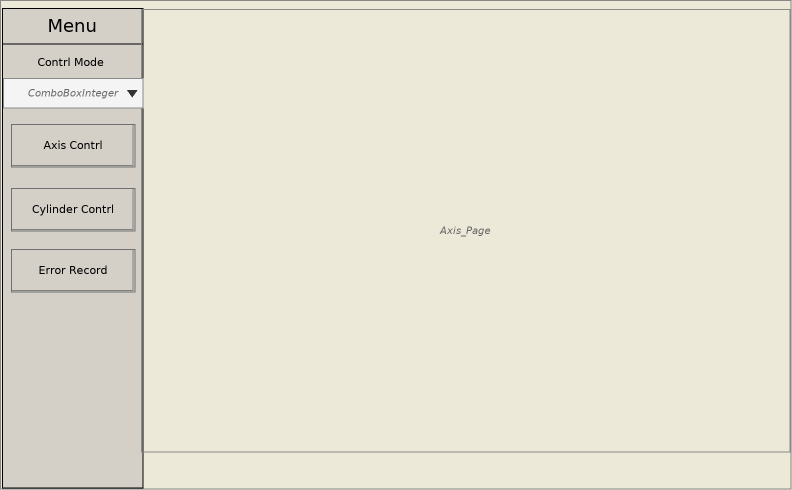
VISUALIZATION Main  // 792x490
    Rectangle (2,8 141x480)
    Rectangle (2,8 141x36), "Menu"
    Rectangle (4,46 134x33), "Contrl Mode"
    Button (11,124 124x43), "Axis Contrl"
        OnMouseDown: FrameSelectionChange Selection=SelectedFrame=54291640-e5ed-4e41-8a36-41169059765e, GlobSel=AssignType=Directly, SelType=Locally
    Button (11,188 124x43), "Cylinder Contrl"
        OnMouseDown: FrameSelectionChange Selection=SelectedFrame=54291640-e5ed-4e41-8a36-41169059765e, Selection=1, GlobSel=AssignType=Directly, SelType=Locally
    Frame (141,9 649x443)
        shows Axis_Page(userdata := gAxisCtrl_HMI[1])
        shows Cylinder(userdata := gCylinderCtrl_HMI[30])
        shows Err_record()
    ComboBoxInteger (3,78 140x30), variable: HMISwithMode, text list: 'CtrlMode_List'
    Button (11,249 124x43), "Error Record"
        OnMouseDown: FrameSelectionChange Selection=SelectedFrame=54291640-e5ed-4e41-8a36-41169059765e, Selection=2, GlobSel=AssignType=Directly, SelType=Locally
END_VISUALIZATION

(* stored: Version 1.1.0.1, ProductVersion 3.1.4018.5
   Visu Main: Id {eb08aa66-22b3-4acc-b5e0-9cb7ae3e017d} *)
